(* PLC project  *)

PROGRAM P
  VAR
    tmr : TON;
  END_VAR

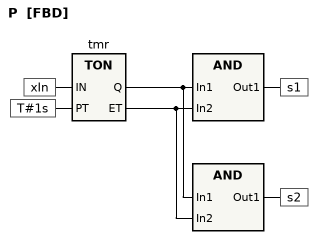
(* FBD diagram, written out as Structured Text *)
tmr(IN := xIn, PT := T#1s);
s1 := tmr.Q AND tmr.ET;
s2 := tmr.Q AND tmr.ET;
END_PROGRAM
